(* Exchanges preemption requests and current beam state with subsystems in arbiter
network.

2019-12-2, A. Wallace

Use in conjunction with FB_SubSysToArbiter_IO.

This FB runs in the beamline arbiter PLC (BAP). There should be one of these for every
subsystem interfaced to the BAP. Each subsystem PLC should run a sibling FB_SubSysToArbiter_IO FB.

This FB and its subordinate communicate through the ethercat connection between the subsystem PLC and the BAP.

A beam parameter set request is sent from the subsystem to this PLC, and includes a cohort number.

This cohort number (i_RequestedBP.nCohortInt) is compared to a local cohort number (nRequestedCohort).
A request from the subsystem to update or modify its current request is indicated by an increase in the
i_RequestedBP.nCohortInt value. Then this function block updates the local arbiter request for the subsystem
and awaits confirmation. Once the new request is confirmed in the preemptive system this function block increments
the ActiveCohort value to match the nRequestedCohort. ActiveCohort is also relayed back to the subsystem
as the active cohort value in the o_CurrentBP set. The subsystem then knows its request has been heard,
and can carry out its own acknowledgement to its various requestors.

Things to note:
If a subsystem has any new or changed preemptive requests you should see the cohort value increment a bit.
If the cohort number is incrementing out of control, it usually means the subsysetm has some preemptive
request loop (two arbiters elevating to each other), or there is a RequestAdd, RequestRemove loop.

*)
FUNCTION_BLOCK FB_ArbiterToSubSys_IO
VAR_INPUT
    RequestingSystemID	:	DWORD := PMPS_GVL.EXCLUDED_ASSERTION_ID; // System ID for making requests to the supreme arbiter
    sName : STRING := 'ArbiterToSubSys';
    Reset : BOOL;
END_VAR
VAR_OUTPUT
END_VAR
VAR_IN_OUT
    Arbiter	: FB_Arbiter;
    fbFFHWO : FB_HardwareFFOutput;
END_VAR
VAR

    i_RequestedBP AT %I*	:	ST_BeamParams_IO; // Requested BP from subsystem
    {attribute 'pytmc' := '
        pv: RequestedBP:FromSubSys
    '}
    RequestedBP: ST_BeamParams;

    o_CurrentBP AT %Q* : ST_BeamParams_IO; // Current BP set

    // EL6692 Diagnostics
    i_Connected AT %I* : BOOL; // SYNC Inputs^External device not connected !!! Doesn't really work.
    {attribute 'pytmc' := 'pv: WcState
        io: i
        field: DESC Working counter state.
        field: ZNAM OK
        field: ONAM Error'}
    i_WcState AT %I* : BOOL := TRUE; // WcState^WcState
    {attribute 'pytmc' := 'pv: TxPDO_state
        io: i
        field: DESC PDO Transmission is OK
        field: ZNAM OK
        field: ONAM Error'}
    i_TxPDOState AT %I* : BOOL := TRUE; // SYNC Inputs^TxPDO state
    {attribute 'pytmc' := 'pv: TxPDO_toggle
        io: i
        field: DESC PDO Transmission is OK
        field: ZNAM OK
        field: ONAM Error'}
    i_TxPDOToggle AT %I* : BOOL; // TxPDO toggle

    // Fast faults
    ffPMPSIO_Disconnect : FB_FastFault := (i_Desc:='Issue w/ arbiter interface to subsystem, verify subsystem is OK, or ethercat connection.'); // Fast fault for ethercat issues
    nActiveCohort : UDINT := 0; // Active cohort. Updated to the req. number from the sub system after request is confirmed.
    nRequestedCohort : UDINT := 0;
    rtToggle : R_TRIG;
    fbToggleTimer : TON;
     tInterval    : TIME := T#100mS;

END_VAR


// Incoming request from subsystem PLC
RequestedBP := IO_TO_BP(i_RequestedBP);

// Update Arbiter with our request
rtToggle(CLK:= i_RequestedBP.xValid); // If interface resumes, reset/catch up
// xValid will go false if the PLC program on the other side is stopped. Ironically the ethercat interface continues happily.
// If subsystem cohort has incremented, update beam parameter request with our arbiter
IF rtToggle.Q THEN
    nActiveCohort := 0;
END_IF

IF i_RequestedBP.nCohortInt > nRequestedCohort OR rtToggle.Q THEN
    Arbiter.RemoveRequest(RequestingSystemID);
    Arbiter.AddRequest(RequestingSystemID, RequestedBP,sName);
    nRequestedCohort := i_RequestedBP.nCohortInt;
END_IF


// Check if latest request is acknowledged by this arbiter
// Acknowledgement happens after an arbitration cycle, which means if RequestedCohort just incremented
// due to a new request, CheckRequest will be false.
IF Arbiter.CheckRequest(RequestingSystemID) THEN
    nActiveCohort := nRequestedCohort; // If it is, then the active cohort is set to the requested cohort number.
END_IF

fbToggleTimer(IN := NOT o_CurrentBP.xValidToggle, PT := tInterval);
// Sending current beam parameter set to subsystems
o_CurrentBP := BP_TO_IO(PMPS_GVL.stCurrentBeamParameters);
o_CurrentBP.nCohortInt := nActiveCohort;
IF (fbToggleTimer.Q) THEN o_CurrentBP.xValidToggle := NOT o_CurrentBP.xValidToggle; END_IF
o_CurrentBP.xValid := TRUE; // This is set and held true here every cycle to prove the PLC on this side is still running


//////////////////////////////////////
// Verifying the ethercat interface health
/////////////////////////////////////
// Both of these values should be 0 for a fully valid exchange
ffPMPSIO_Disconnect.i_xOK := NOT i_WcState AND NOT i_TxPDOState;

ffPMPSIO_Disconnect(
    io_fbFFHWO := fbFFHWO,
    i_xReset := Reset,
    i_DevName := sName,
    i_TypeCode:=5);

END_FUNCTION_BLOCK

(* stored: Version 1.1.0.1
   POU FB_ArbiterToSubSys_IO: Id {1a7d9761-dced-4384-823d-a5e0b037bf80}, SpecialFunc None *)
